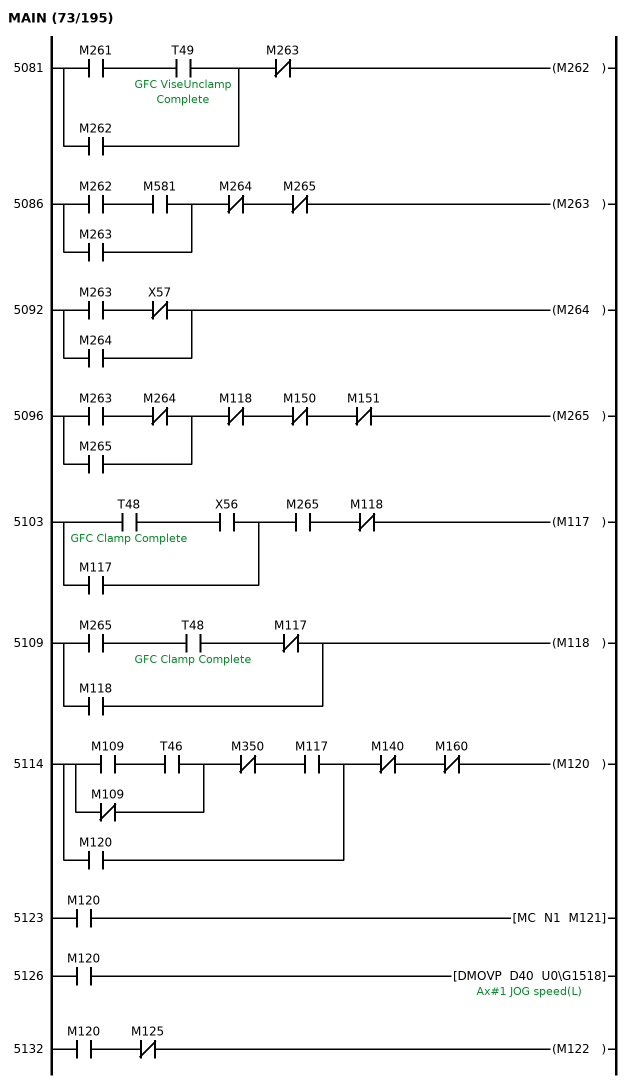
[picture p72: ladder of MAIN, rungs at steps 5081 to 5132]
5081  LD      M261
      AND     T49  ; GFC ViseUnclamp Complete
      OR      M262
      ANI     M263
      OUT     M262
5086  LD      M262
      AND     M581
      OR      M263
      ANI     M264
      ANI     M265
      OUT     M263
5092  LD      M263
      ANI     X57
      OR      M264
      OUT     M264
5096  LD      M263
      ANI     M264
      OR      M265
      ANI     M118
      ANI     M150
      ANI     M151
      OUT     M265
5103  LD      T48  ; GFC Clamp Complete
      AND     X56
      OR      M117
      AND     M265
      ANI     M118
      OUT     M117
5109  LD      M265
      AND     T48  ; GFC Clamp Complete
      ANI     M117
      OR      M118
      OUT     M118
5114  LD      M109
      AND     T46
      ORI     M109
      ANI     M350
      AND     M117
      OR      M120
      ANI     M140
      ANI     M160
      OUT     M120
5123  LD      M120
      MC      N1 M121
5126  LD      M120
      DMOVP   D40 U0\G1518
5132  LD      M120
      ANI     M125
      OUT     M122
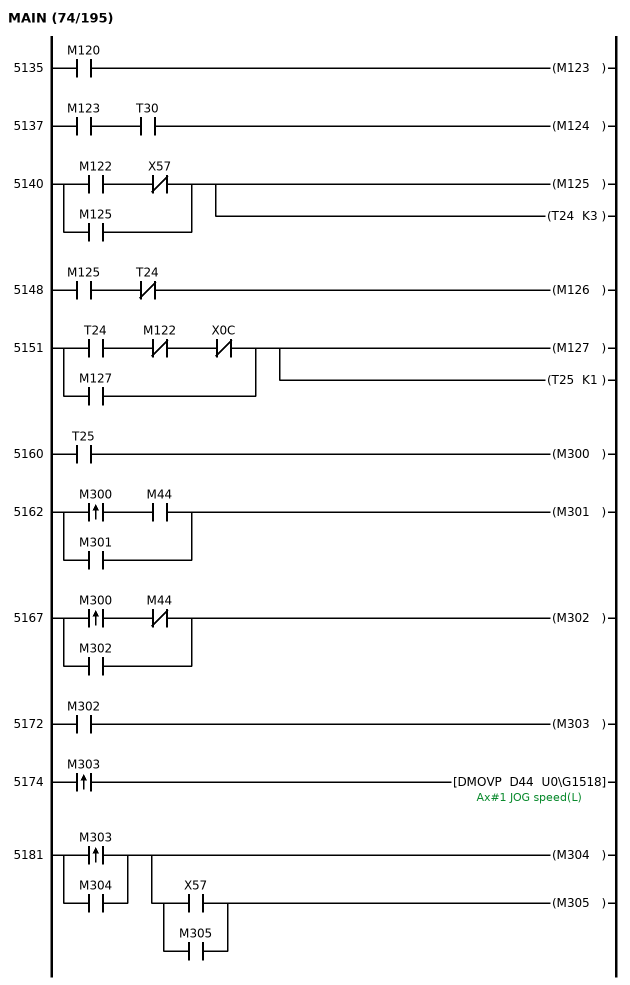
5135  LD      M120
      OUT     M123
5137  LD      M123
      AND     T30
      OUT     M124
5140  LD      M122
      ANI     X57
      OR      M125
      OUT     M125
      OUT     T24 K3
5148  LD      M125
      ANI     T24
      OUT     M126
5151  LD      T24
      ANI     M122
      ANI     X0C
      OR      M127
      OUT     M127
      OUT     T25 K1
5160  LD      T25
      OUT     M300
5162  LDP     M300
      AND     M44
      OR      M301
      OUT     M301
5167  LDP     M300
      ANI     M44
      OR      M302
      OUT     M302
5172  LD      M302
      OUT     M303
5174  LDP     M303
      DMOVP   D44 U0\G1518
5181  LDP     M303
      OR      M304
      OUT     M304
      LD      X57
      OR      M305
      ANB
      OUT     M305
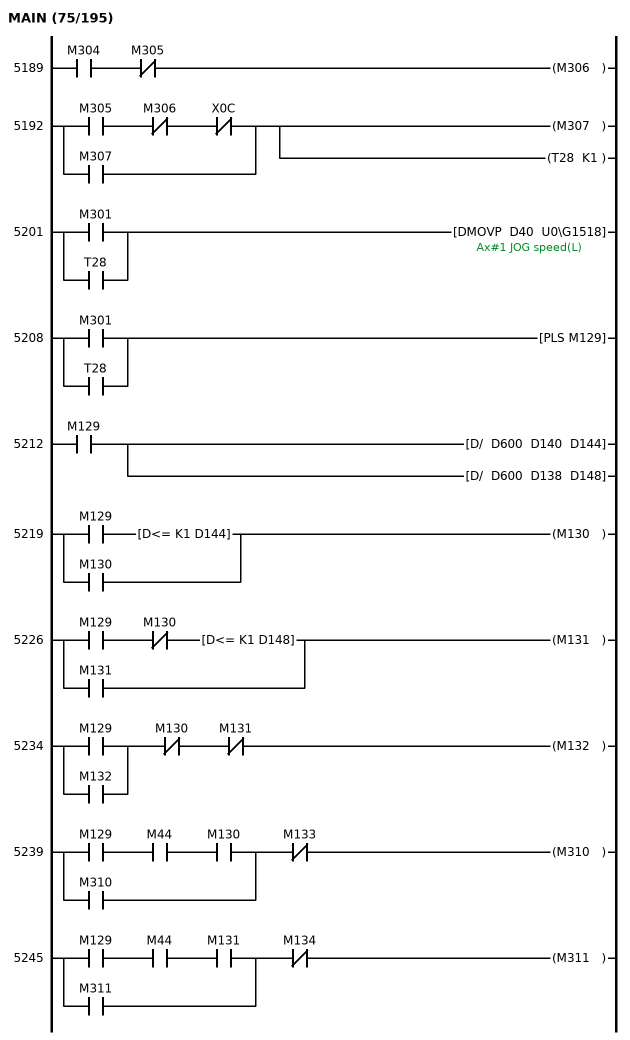
5189  LD      M304
      ANI     M305
      OUT     M306
5192  LD      M305
      ANI     M306
      ANI     X0C
      OR      M307
      OUT     M307
      OUT     T28 K1
5201  LD      M301
      OR      T28
      DMOVP   D40 U0\G1518
5208  LD      M301
      OR      T28
      PLS     M129
5212  LD      M129
      D/      D600 D140 D144
      D/      D600 D138 D148
5219  LD      M129
      ANDD<=  K1 D144
      OR      M130
      OUT     M130
5226  LD      M129
      ANI     M130
      ANDD<=  K1 D148
      OR      M131
      OUT     M131
5234  LD      M129
      OR      M132
      ANI     M130
      ANI     M131
      OUT     M132
5239  LD      M129
      AND     M44
      AND     M130
      OR      M310
      ANI     M133
      OUT     M310
5245  LD      M129
      AND     M44
      AND     M131
      OR      M311
      ANI     M134
      OUT     M311
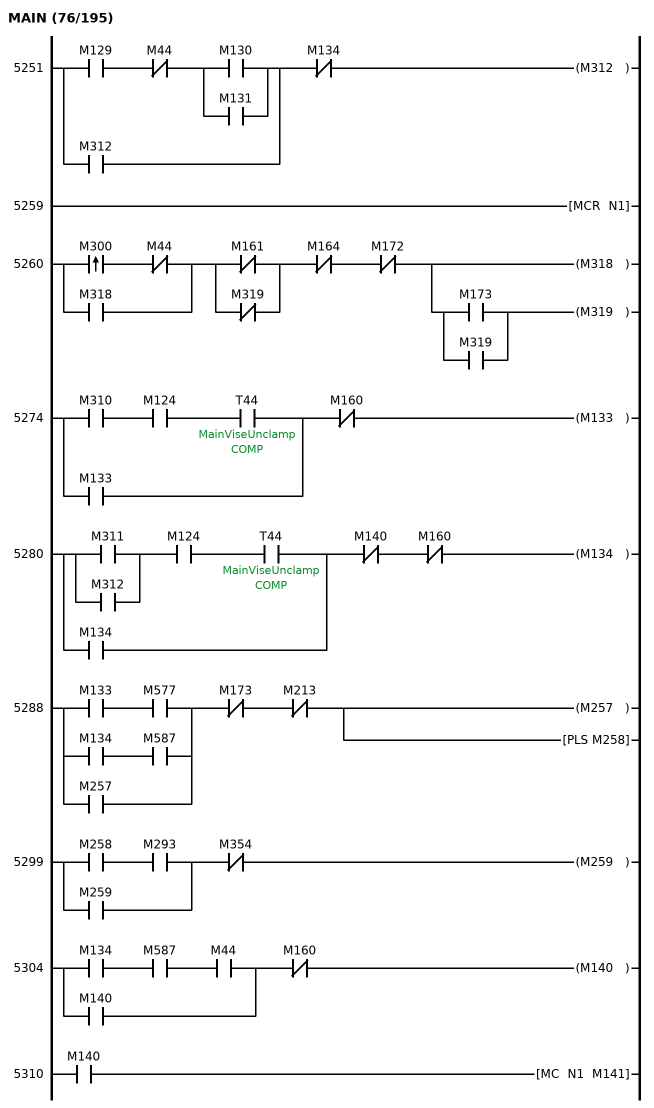
5251  LD      M129
      ANI     M44
      LD      M130
      OR      M131
      ANB
      OR      M312
      ANI     M134
      OUT     M312
5259  MCR     N1
5260  LDP     M300
      ANI     M44
      OR      M318
      LDI     M161
      ORI     M319
      ANB
      ANI     M164
      ANI     M172
      OUT     M318
      LD      M173
      OR      M319
      ANB
      OUT     M319
5274  LD      M310
      AND     M124
      AND     T44  ; MainViseUnclamp COMP
      OR      M133
      ANI     M160
      OUT     M133
5280  LD      M311
      OR      M312
      AND     M124
      AND     T44  ; MainViseUnclamp COMP
      OR      M134
      ANI     M140
      ANI     M160
      OUT     M134
5288  LD      M133
      AND     M577
      LD      M134
      AND     M587
      ORB
      OR      M257
      ANI     M173
      ANI     M213
      OUT     M257
      PLS     M258
5299  LD      M258
      AND     M293
      OR      M259
      ANI     M354
      OUT     M259
5304  LD      M134
      AND     M587
      AND     M44
      OR      M140
      ANI     M160
      OUT     M140
5310  LD      M140
      MC      N1 M141
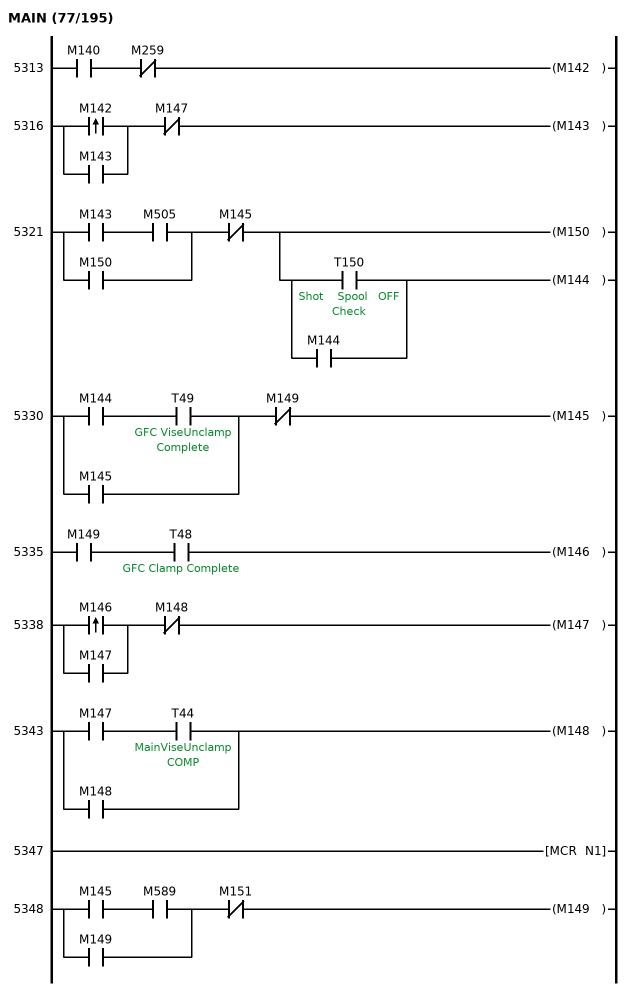
5313  LD      M140
      ANI     M259
      OUT     M142
5316  LDP     M142
      OR      M143
      ANI     M147
      OUT     M143
5321  LD      M143
      AND     M505
      OR      M150
      ANI     M145
      OUT     M150
      LD      T150  ; Shot    Spool   OFF     Check
      OR      M144
      ANB
      OUT     M144
5330  LD      M144
      AND     T49  ; GFC ViseUnclamp Complete
      OR      M145
      ANI     M149
      OUT     M145
5335  LD      M149
      AND     T48  ; GFC Clamp Complete
      OUT     M146
5338  LDP     M146
      OR      M147
      ANI     M148
      OUT     M147
5343  LD      M147
      AND     T44  ; MainViseUnclamp COMP
      OR      M148
      OUT     M148
5347  MCR     N1
5348  LD      M145
      AND     M589
      OR      M149
      ANI     M151
      OUT     M149
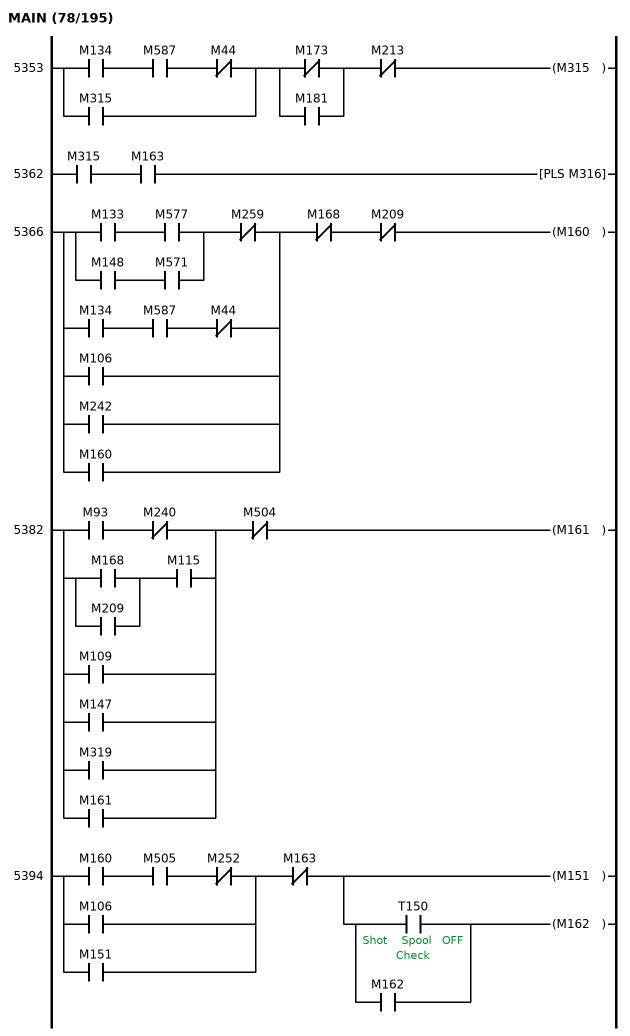
5353  LD      M134
      AND     M587
      ANI     M44
      OR      M315
      LDI     M173
      OR      M181
      ANB
      ANI     M213
      OUT     M315
5362  LD      M315
      AND     M163
      PLS     M316
5366  LD      M133
      AND     M577
      LD      M148
      AND     M571
      ORB
      ANI     M259
      LD      M134
      AND     M587
      ANI     M44
      ORB
      OR      M106
      OR      M242
      OR      M160
      ANI     M168
      ANI     M209
      OUT     M160
5382  LD      M93
      ANI     M240
      LD      M168
      OR      M209
      AND     M115
      ORB
      OR      M109
      OR      M147
      OR      M319
      OR      M161
      ANI     M504
      OUT     M161
5394  LD      M160
      AND     M505
      ANI     M252
      OR      M106
      OR      M151
      ANI     M163
      OUT     M151
      LD      T150  ; Shot    Spool   OFF     Check
      OR      M162
      ANB
      OUT     M162
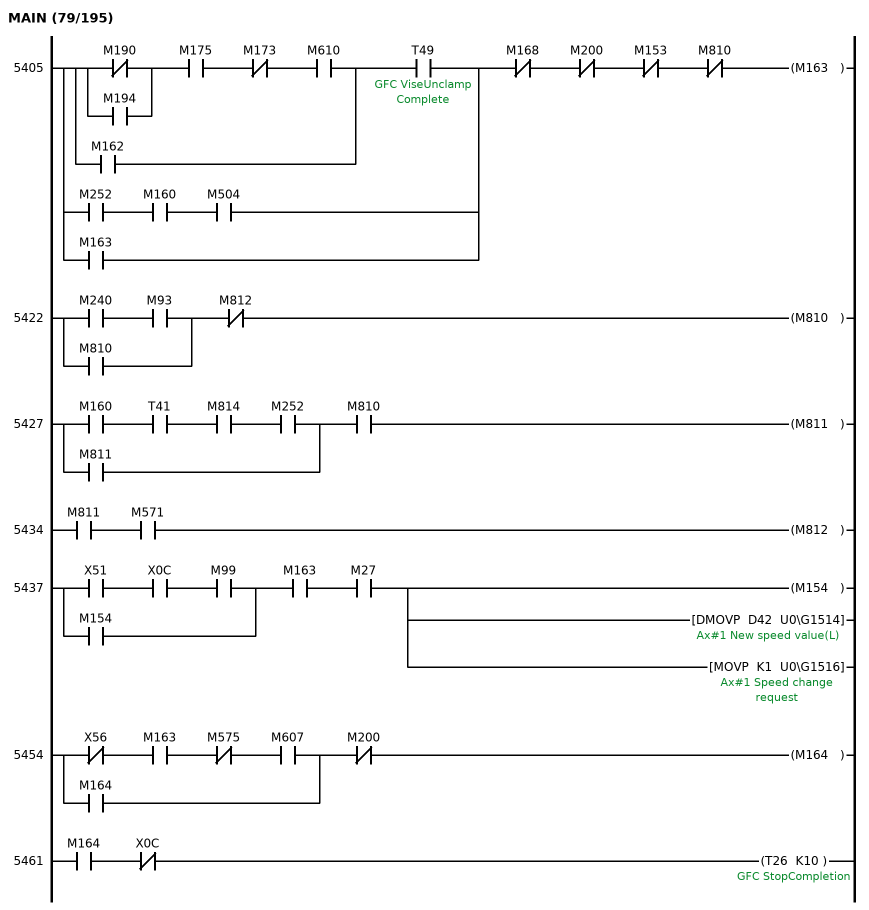
5405  LDI     M190
      OR      M194
      AND     M175
      ANI     M173
      AND     M610
      OR      M162
      AND     T49  ; GFC ViseUnclamp Complete
      LD      M252
      AND     M160
      AND     M504
      ORB
      OR      M163
      ANI     M168
      ANI     M200
      ANI     M153
      ANI     M810
      OUT     M163
5422  LD      M240
      AND     M93
      OR      M810
      ANI     M812
      OUT     M810
5427  LD      M160
      AND     T41
      AND     M814
      AND     M252
      OR      M811
      AND     M810
      OUT     M811
5434  LD      M811
      AND     M571
      OUT     M812
5437  LD      X51
      AND     X0C
      AND     M99
      OR      M154
      AND     M163
      AND     M27
      OUT     M154
      DMOVP   D42 U0\G1514  ; Ax#1 New speed value(L)
      MOVP    K1 U0\G1516  ; Ax#1 Speed change request
5454  LDI     X56
      AND     M163
      ANI     M575
      AND     M607
      OR      M164
      ANI     M200
      OUT     M164
5461  LD      M164
      ANI     X0C
      OUT     T26 K10  ; GFC StopCompletion
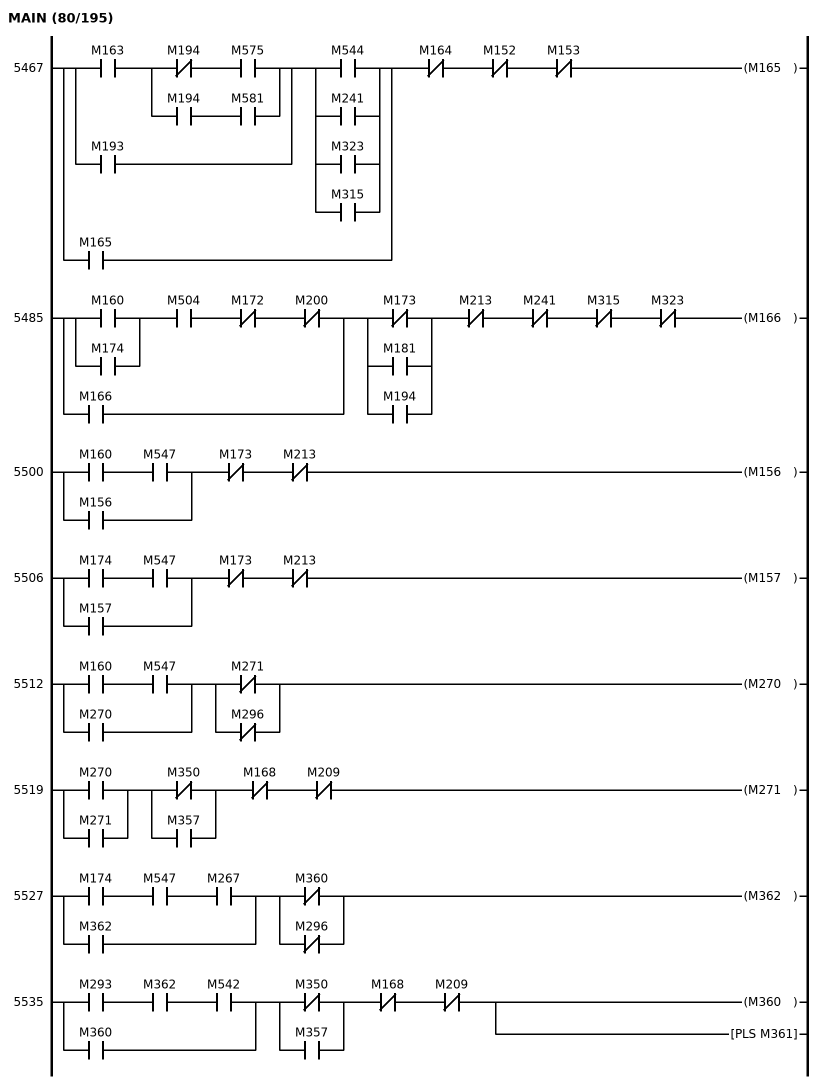
5467  LD      M163
      LDI     M194
      AND     M575
      LD      M194
      AND     M581
      ORB
      ANB
      OR      M193
      LD      M544
      OR      M241
      OR      M323
      OR      M315
      ANB
      OR      M165
      ANI     M164
      ANI     M152
      ANI     M153
      OUT     M165
5485  LD      M160
      OR      M174
      AND     M504
      ANI     M172
      ANI     M200
      OR      M166
      LDI     M173
      OR      M181
      OR      M194
      ANB
      ANI     M213
      ANI     M241
      ANI     M315
      ANI     M323
      OUT     M166
5500  LD      M160
      AND     M547
      OR      M156
      ANI     M173
      ANI     M213
      OUT     M156
5506  LD      M174
      AND     M547
      OR      M157
      ANI     M173
      ANI     M213
      OUT     M157
5512  LD      M160
      AND     M547
      OR      M270
      LDI     M271
      ORI     M296
      ANB
      OUT     M270
5519  LD      M270
      OR      M271
      LDI     M350
      OR      M357
      ANB
      ANI     M168
      ANI     M209
      OUT     M271
5527  LD      M174
      AND     M547
      AND     M267
      OR      M362
      LDI     M360
      ORI     M296
      ANB
      OUT     M362
5535  LD      M293
      AND     M362
      AND     M542
      OR      M360
      LDI     M350
      OR      M357
      ANB
      ANI     M168
      ANI     M209
      OUT     M360
      PLS     M361
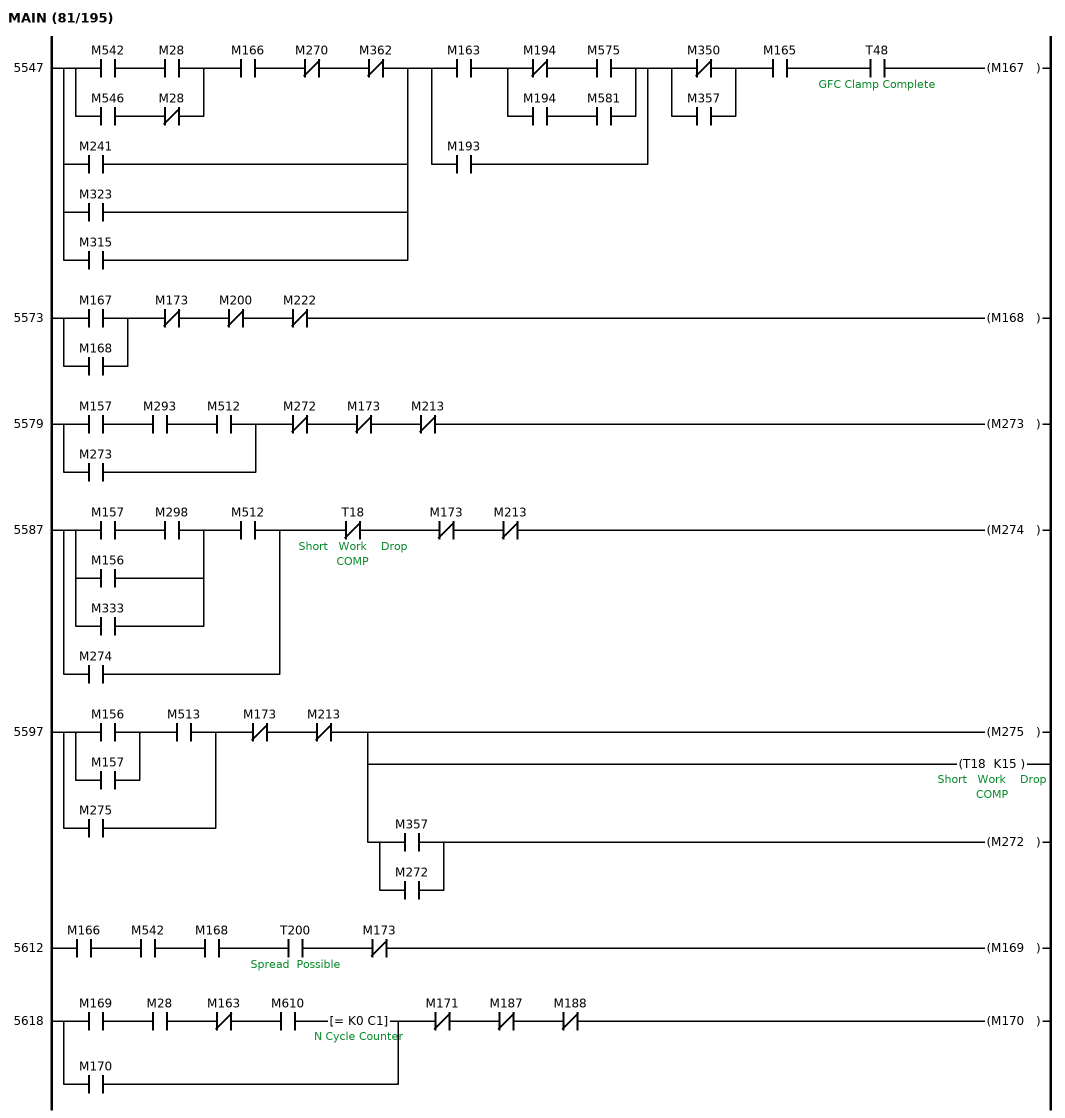
5547  LD      M542
      AND     M28
      LD      M546
      ANI     M28
      ORB
      AND     M166
      ANI     M270
      ANI     M362
      OR      M241
      OR      M323
      OR      M315
      LD      M163
      LDI     M194
      AND     M575
      LD      M194
      AND     M581
      ORB
      ANB
      OR      M193
      ANB
      LDI     M350
      OR      M357
      ANB
      AND     M165
      AND     T48  ; GFC Clamp Complete
      OUT     M167
5573  LD      M167
      OR      M168
      ANI     M173
      ANI     M200
      ANI     M222
      OUT     M168
5579  LD      M157
      AND     M293
      AND     M512
      OR      M273
      ANI     M272
      ANI     M173
      ANI     M213
      OUT     M273
5587  LD      M157
      AND     M298
      OR      M156
      OR      M333
      AND     M512
      OR      M274
      ANI     T18  ; Short   Work    Drop    COMP
      ANI     M173
      ANI     M213
      OUT     M274
5597  LD      M156
      OR      M157
      AND     M513
      OR      M275
      ANI     M173
      ANI     M213
      OUT     M275
      OUT     T18 K15  ; Short   Work    Drop    COMP
      LD      M357
      OR      M272
      ANB
      OUT     M272
5612  LD      M166
      AND     M542
      AND     M168
      AND     T200  ; Spread  Possible
      ANI     M173
      OUT     M169
5618  LD      M169
      AND     M28
      ANI     M163
      AND     M610
      AND=    K0 C1  ; N Cycle Counter
      OR      M170
      ANI     M171
      ANI     M187
      ANI     M188
      OUT     M170
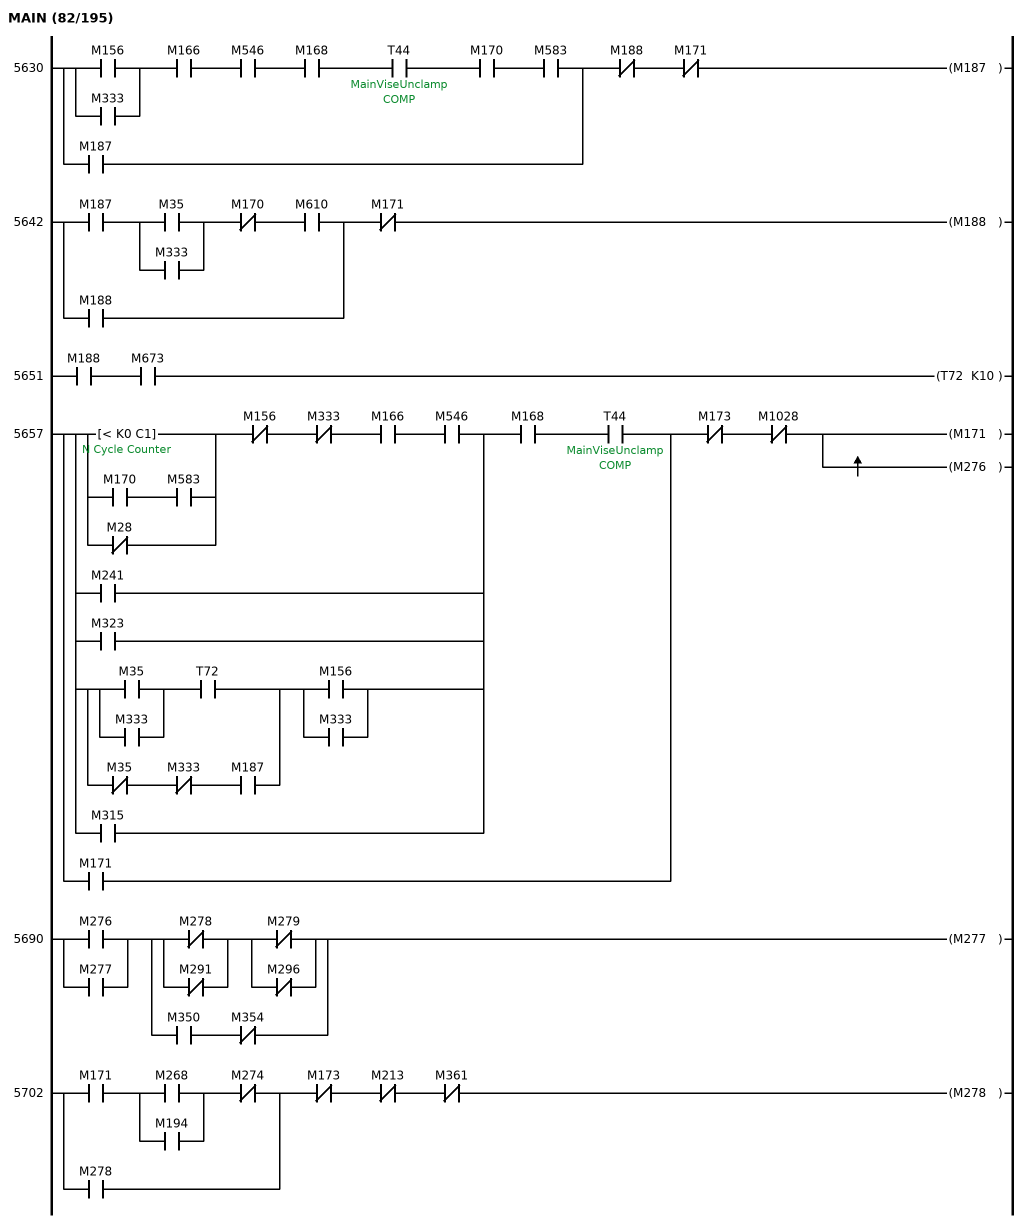
5630  LD      M156
      OR      M333
      AND     M166
      AND     M546
      AND     M168
      AND     T44  ; MainViseUnclamp COMP
      AND     M170
      AND     M583
      OR      M187
      ANI     M188
      ANI     M171
      OUT     M187
5642  LD      M187
      LD      M35
      OR      M333
      ANB
      ANI     M170
      AND     M610
      OR      M188
      ANI     M171
      OUT     M188
5651  LD      M188
      AND     M673
      OUT     T72 K10
5657  LD<     K0 C1  ; N Cycle Counter
      LD      M170
      AND     M583
      ORB
      ORI     M28
      ANI     M156
      ANI     M333
      AND     M166
      AND     M546
      OR      M241
      OR      M323
      LD      M35
      OR      M333
      AND     T72
      LDI     M35
      ANI     M333
      AND     M187
      ORB
      LD      M156
      OR      M333
      ANB
      ORB
      OR      M315
      AND     M168
      AND     T44  ; MainViseUnclamp COMP
      OR      M171
      ANI     M173
      ANI     M1028
      OUT     M171
      MEP
      OUT     M276
5690  LD      M276
      OR      M277
      LDI     M278
      ORI     M291
      LDI     M279
      ORI     M296
      ANB
      LD      M350
      ANI     M354
      ORB
      ANB
      OUT     M277
5702  LD      M171
      LD      M268
      OR      M194
      ANB
      ANI     M274
      OR      M278
      ANI     M173
      ANI     M213
      ANI     M361
      OUT     M278
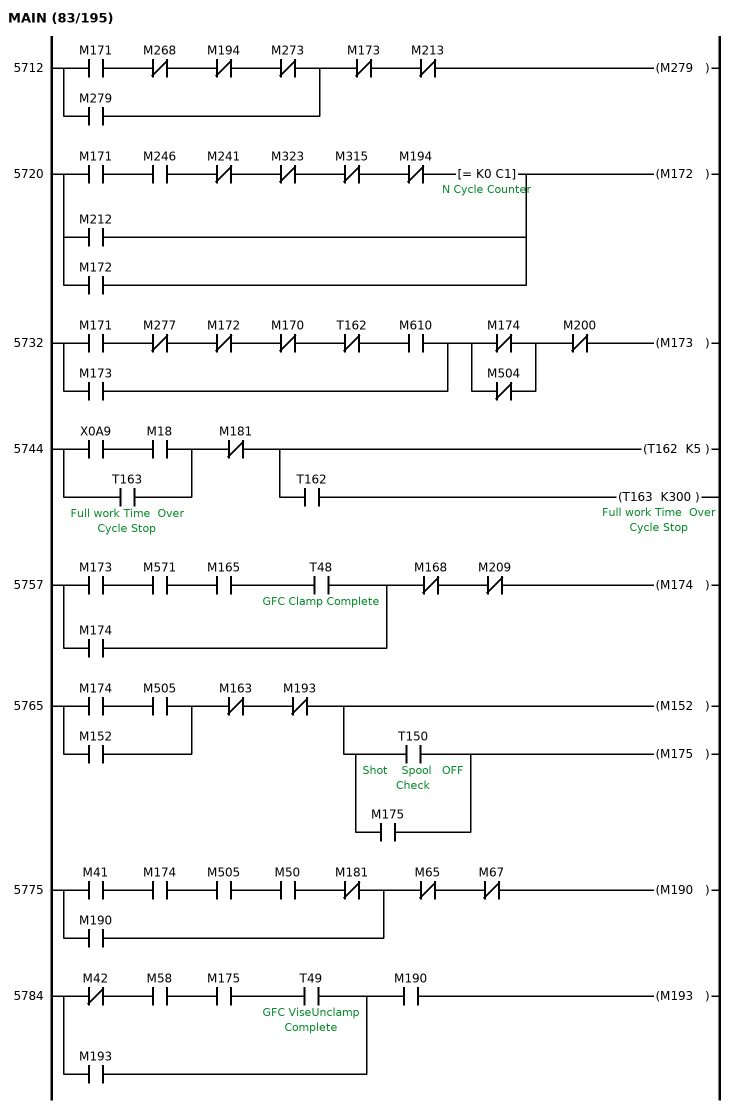
5712  LD      M171
      ANI     M268
      ANI     M194
      ANI     M273
      OR      M279
      ANI     M173
      ANI     M213
      OUT     M279
5720  LD      M171
      AND     M246
      ANI     M241
      ANI     M323
      ANI     M315
      ANI     M194
      AND=    K0 C1  ; N Cycle Counter
      OR      M212
      OR      M172
      OUT     M172
5732  LD      M171
      ANI     M277
      ANI     M172
      ANI     M170
      ANI     T162
      AND     M610
      OR      M173
      LDI     M174
      ORI     M504
      ANB
      ANI     M200
      OUT     M173
5744  LD      X0A9
      AND     M18
      OR      T163  ; Full work Time  Over Cycle Stop
      ANI     M181
      OUT     T162 K5
      AND     T162
      OUT     T163 K300  ; Full work Time  Over Cycle Stop
5757  LD      M173
      AND     M571
      AND     M165
      AND     T48  ; GFC Clamp Complete
      OR      M174
      ANI     M168
      ANI     M209
      OUT     M174
5765  LD      M174
      AND     M505
      OR      M152
      ANI     M163
      ANI     M193
      OUT     M152
      LD      T150  ; Shot    Spool   OFF     Check
      OR      M175
      ANB
      OUT     M175
5775  LD      M41
      AND     M174
      AND     M505
      AND     M50
      ANI     M181
      OR      M190
      ANI     M65
      ANI     M67
      OUT     M190
5784  LDI     M42
      AND     M58
      AND     M175
      AND     T49  ; GFC ViseUnclamp Complete
      OR      M193
      AND     M190
      OUT     M193
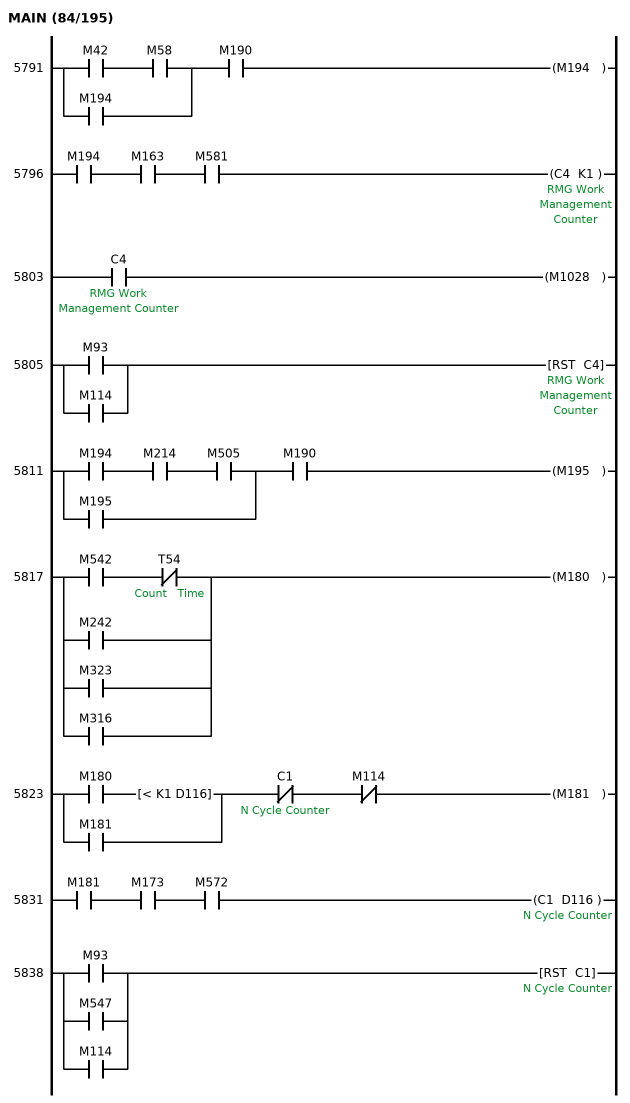
5791  LD      M42
      AND     M58
      OR      M194
      AND     M190
      OUT     M194
5796  LD      M194
      AND     M163
      AND     M581
      OUT     C4 K1  ; RMG WorkManagement Counter
5803  LD      C4  ; RMG WorkManagement Counter
      OUT     M1028
5805  LD      M93
      OR      M114
      RST     C4  ; RMG WorkManagement Counter
5811  LD      M194
      AND     M214
      AND     M505
      OR      M195
      AND     M190
      OUT     M195
5817  LD      M542
      ANI     T54  ; Count   Time
      OR      M242
      OR      M323
      OR      M316
      OUT     M180
5823  LD      M180
      AND<    K1 D116
      OR      M181
      ANI     C1  ; N Cycle Counter
      ANI     M114
      OUT     M181
5831  LD      M181
      AND     M173
      AND     M572
      OUT     C1 D116  ; N Cycle Counter
5838  LD      M93
      OR      M547
      OR      M114
      RST     C1  ; N Cycle Counter
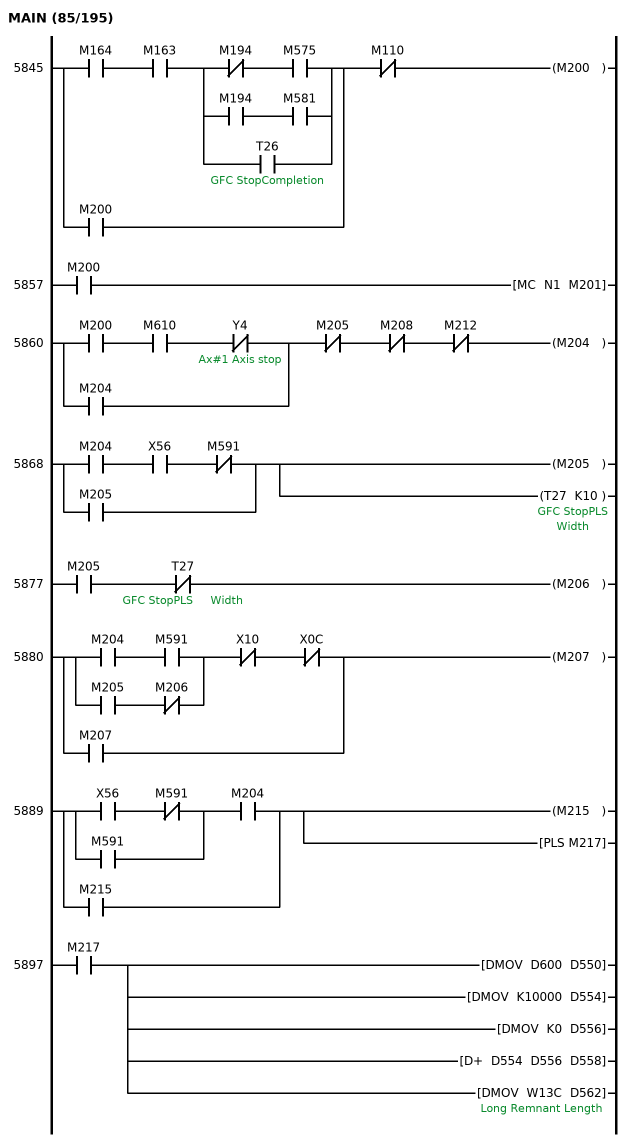
5845  LD      M164
      AND     M163
      LDI     M194
      AND     M575
      LD      M194
      AND     M581
      ORB
      OR      T26  ; GFC StopCompletion
      ANB
      OR      M200
      ANI     M110
      OUT     M200
5857  LD      M200
      MC      N1 M201
5860  LD      M200
      AND     M610
      ANI     Y4  ; Ax#1 Axis stop
      OR      M204
      ANI     M205
      ANI     M208
      ANI     M212
      OUT     M204
5868  LD      M204
      AND     X56
      ANI     M591
      OR      M205
      OUT     M205
      OUT     T27 K10  ; GFC StopPLS     Width
5877  LD      M205
      ANI     T27  ; GFC StopPLS     Width
      OUT     M206
5880  LD      M204
      AND     M591
      LD      M205
      ANI     M206
      ORB
      ANI     X10
      ANI     X0C
      OR      M207
      OUT     M207
5889  LD      X56
      ANI     M591
      OR      M591
      AND     M204
      OR      M215
      OUT     M215
      PLS     M217
5897  LD      M217
      DMOV    D600 D550
      DMOV    K10000 D554
      DMOV    K0 D556
      D+      D554 D556 D558
      DMOV    W13C D562  ; Long Remnant Length
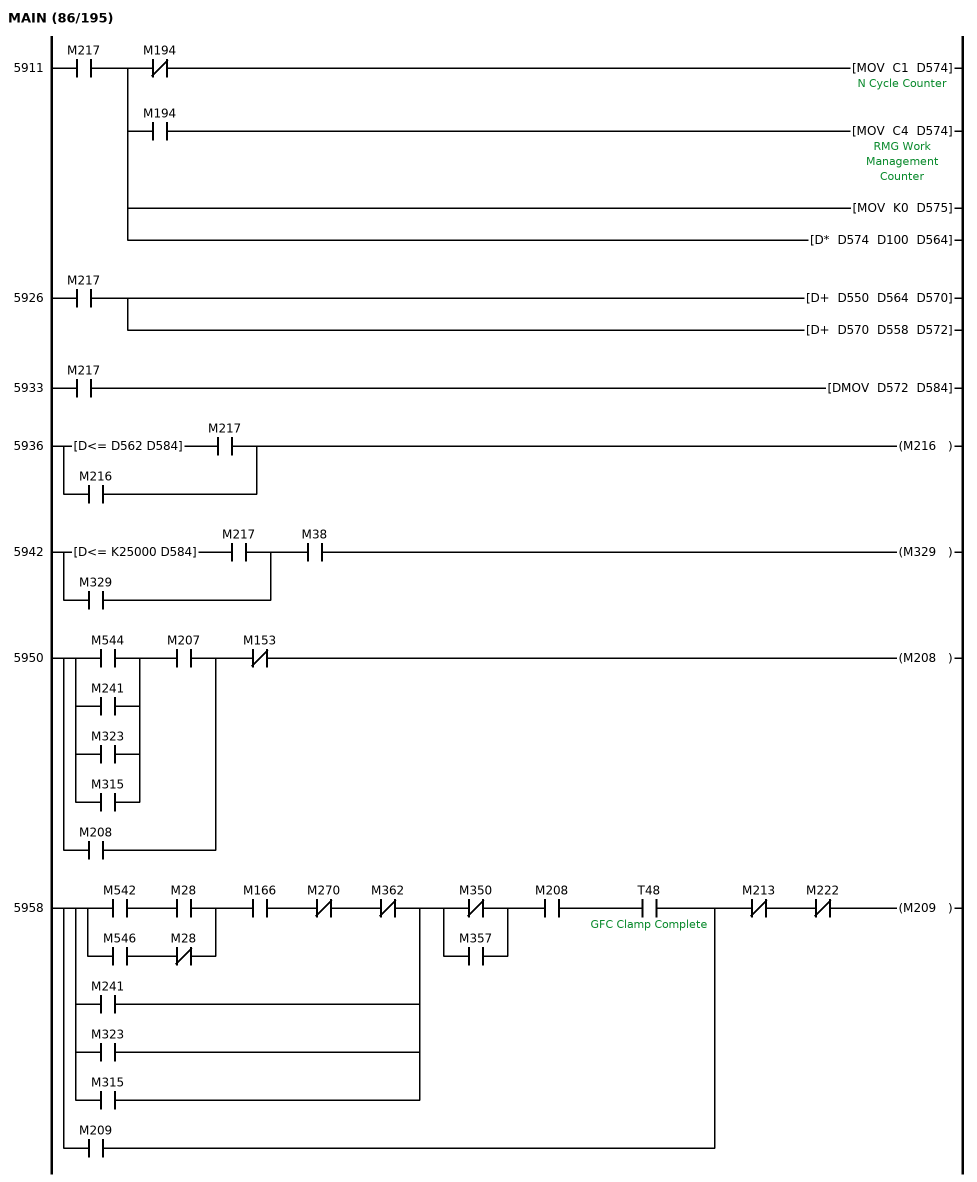
5911  LD      M217
      MPS
      ANI     M194
      MOV     C1 D574
      MRD
      AND     M194
      MOV     C4 D574
      MPP
      MOV     K0 D575
      D*      D574 D100 D564
5926  LD      M217
      D+      D550 D564 D570
      D+      D570 D558 D572
5933  LD      M217
      DMOV    D572 D584
5936  LDD<=   D562 D584
      AND     M217
      OR      M216
      OUT     M216
5942  LDD<=   K25000 D584
      AND     M217
      OR      M329
      AND     M38
      OUT     M329
5950  LD      M544
      OR      M241
      OR      M323
      OR      M315
      AND     M207
      OR      M208
      ANI     M153
      OUT     M208
5958  LD      M542
      AND     M28
      LD      M546
      ANI     M28
      ORB
      AND     M166
      ANI     M270
      ANI     M362
      OR      M241
      OR      M323
      OR      M315
      LDI     M350
      OR      M357
      ANB
      AND     M208
      AND     T48  ; GFC Clamp Complete
      OR      M209
      ANI     M213
      ANI     M222
      OUT     M209
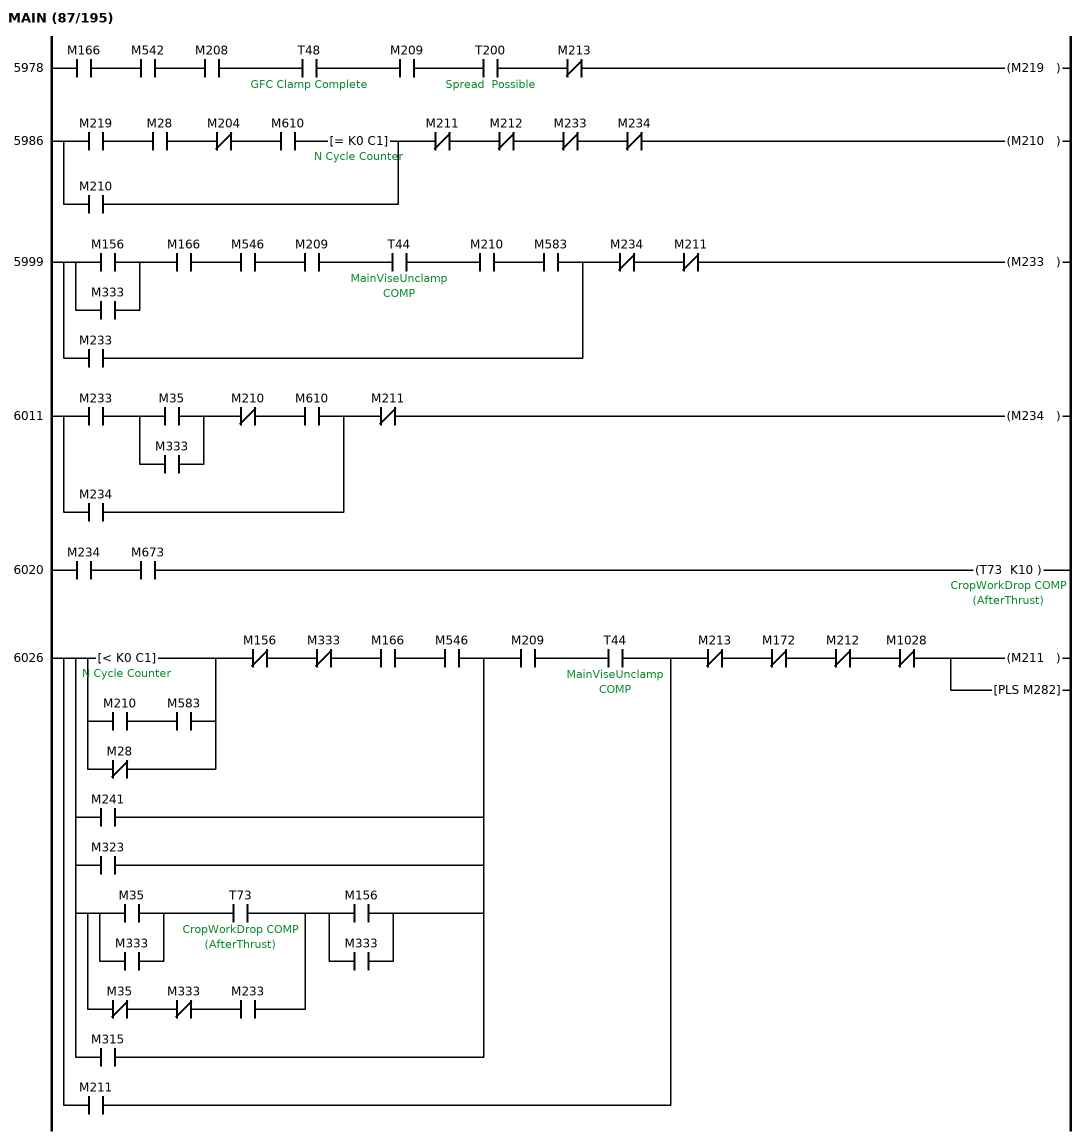
5978  LD      M166
      AND     M542
      AND     M208
      AND     T48  ; GFC Clamp Complete
      AND     M209
      AND     T200  ; Spread  Possible
      ANI     M213
      OUT     M219
5986  LD      M219
      AND     M28
      ANI     M204
      AND     M610
      AND=    K0 C1  ; N Cycle Counter
      OR      M210
      ANI     M211
      ANI     M212
      ANI     M233
      ANI     M234
      OUT     M210
5999  LD      M156
      OR      M333
      AND     M166
      AND     M546
      AND     M209
      AND     T44  ; MainViseUnclamp COMP
      AND     M210
      AND     M583
      OR      M233
      ANI     M234
      ANI     M211
      OUT     M233
6011  LD      M233
      LD      M35
      OR      M333
      ANB
      ANI     M210
      AND     M610
      OR      M234
      ANI     M211
      OUT     M234
6020  LD      M234
      AND     M673
      OUT     T73 K10  ; CropWorkDrop COMP (AfterThrust)
6026  LD<     K0 C1  ; N Cycle Counter
      LD      M210
      AND     M583
      ORB
      ORI     M28
      ANI     M156
      ANI     M333
      AND     M166
      AND     M546
      OR      M241
      OR      M323
      LD      M35
      OR      M333
      AND     T73  ; CropWorkDrop COMP (AfterThrust)
      LDI     M35
      ANI     M333
      AND     M233
      ORB
      LD      M156
      OR      M333
      ANB
      ORB
      OR      M315
      AND     M209
      AND     T44  ; MainViseUnclamp COMP
      OR      M211
      ANI     M213
      ANI     M172
      ANI     M212
      ANI     M1028
      OUT     M211
      PLS     M282
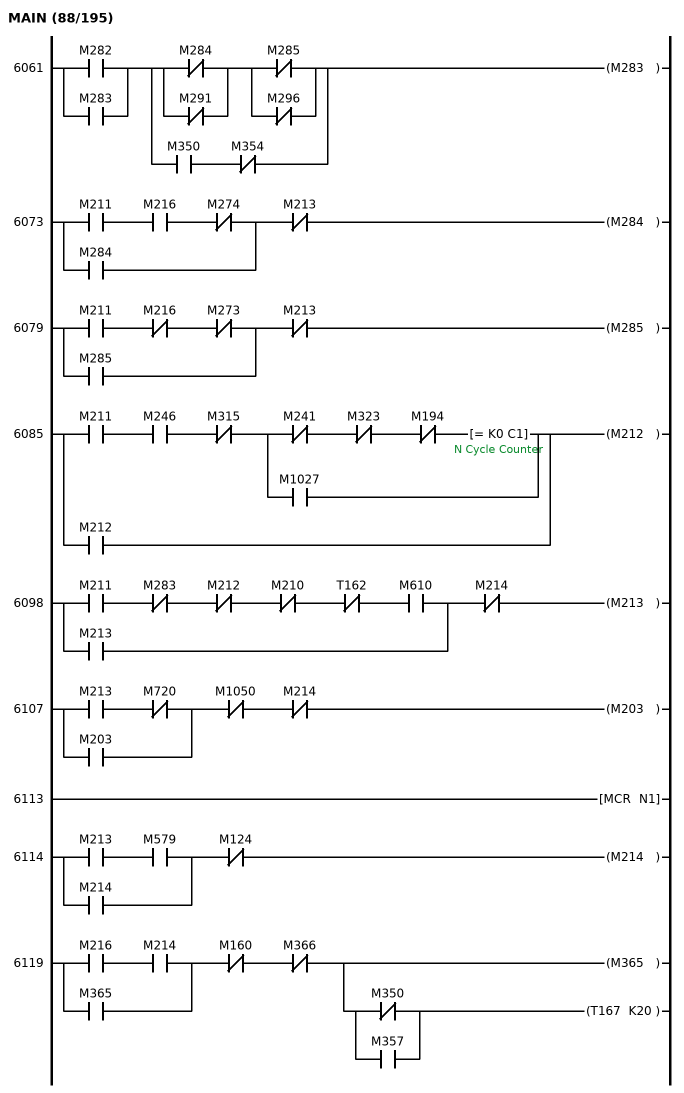
6061  LD      M282
      OR      M283
      LDI     M284
      ORI     M291
      LDI     M285
      ORI     M296
      ANB
      LD      M350
      ANI     M354
      ORB
      ANB
      OUT     M283
6073  LD      M211
      AND     M216
      ANI     M274
      OR      M284
      ANI     M213
      OUT     M284
6079  LD      M211
      ANI     M216
      ANI     M273
      OR      M285
      ANI     M213
      OUT     M285
6085  LD      M211
      AND     M246
      ANI     M315
      LDI     M241
      ANI     M323
      ANI     M194
      AND=    K0 C1  ; N Cycle Counter
      OR      M1027
      ANB
      OR      M212
      OUT     M212
6098  LD      M211
      ANI     M283
      ANI     M212
      ANI     M210
      ANI     T162
      AND     M610
      OR      M213
      ANI     M214
      OUT     M213
6107  LD      M213
      ANI     M720
      OR      M203
      ANI     M1050
      ANI     M214
      OUT     M203
6113  MCR     N1
6114  LD      M213
      AND     M579
      OR      M214
      ANI     M124
      OUT     M214
6119  LD      M216
      AND     M214
      OR      M365
      ANI     M160
      ANI     M366
      OUT     M365
      LDI     M350
      OR      M357
      ANB
      OUT     T167 K20
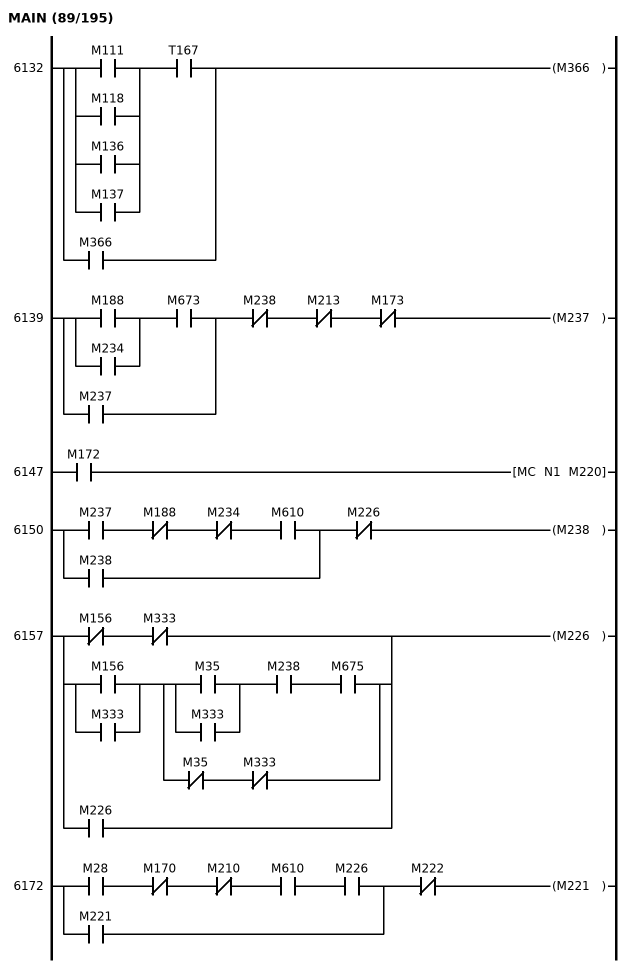
6132  LD      M111
      OR      M118
      OR      M136
      OR      M137
      AND     T167
      OR      M366
      OUT     M366
6139  LD      M188
      OR      M234
      AND     M673
      OR      M237
      ANI     M238
      ANI     M213
      ANI     M173
      OUT     M237
6147  LD      M172
      MC      N1 M220
6150  LD      M237
      ANI     M188
      ANI     M234
      AND     M610
      OR      M238
      ANI     M226
      OUT     M238
6157  LDI     M156
      ANI     M333
      LD      M156
      OR      M333
      LD      M35
      OR      M333
      AND     M238
      AND     M675
      LDI     M35
      ANI     M333
      ORB
      ANB
      ORB
      OR      M226
      OUT     M226
6172  LD      M28
      ANI     M170
      ANI     M210
      AND     M610
      AND     M226
      OR      M221
      ANI     M222
      OUT     M221
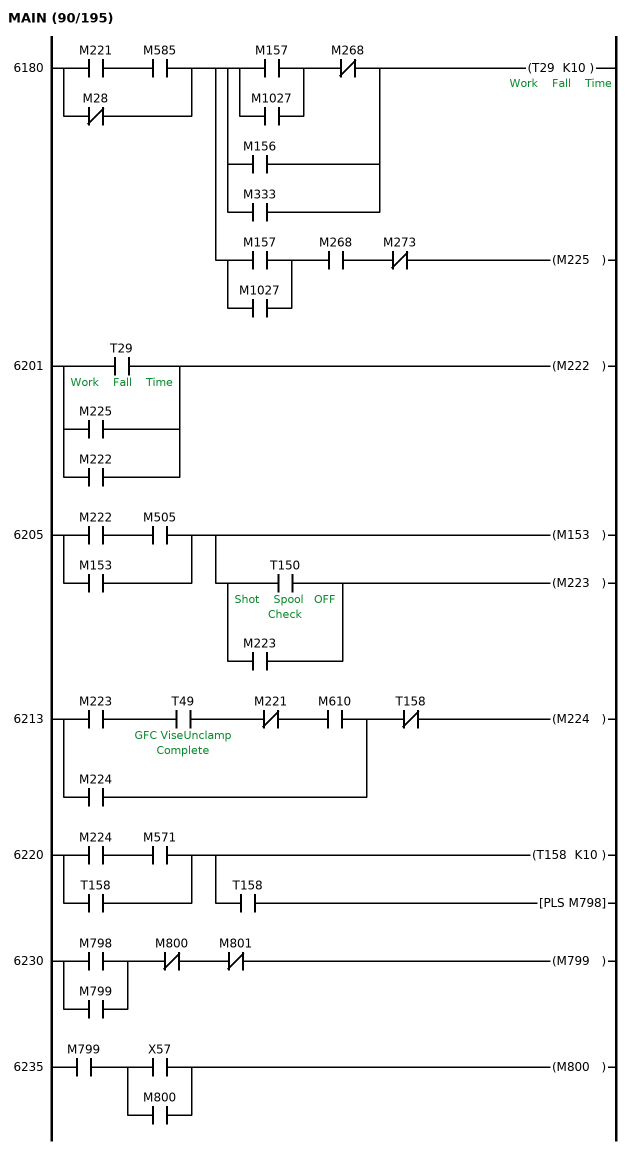
6180  LD      M221
      AND     M585
      ORI     M28
      MPS
      LD      M157
      OR      M1027
      ANI     M268
      OR      M156
      OR      M333
      ANB
      OUT     T29 K10  ; Work    Fall    Time
      MPP
      LD      M157
      OR      M1027
      ANB
      AND     M268
      ANI     M273
      OUT     M225
6201  LD      T29  ; Work    Fall    Time
      OR      M225
      OR      M222
      OUT     M222
6205  LD      M222
      AND     M505
      OR      M153
      OUT     M153
      LD      T150  ; Shot    Spool   OFF     Check
      OR      M223
      ANB
      OUT     M223
6213  LD      M223
      AND     T49  ; GFC ViseUnclamp Complete
      ANI     M221
      AND     M610
      OR      M224
      ANI     T158
      OUT     M224
6220  LD      M224
      AND     M571
      OR      T158
      OUT     T158 K10
      AND     T158
      PLS     M798
6230  LD      M798
      OR      M799
      ANI     M800
      ANI     M801
      OUT     M799
6235  LD      M799
      LD      X57
      OR      M800
      ANB
      OUT     M800
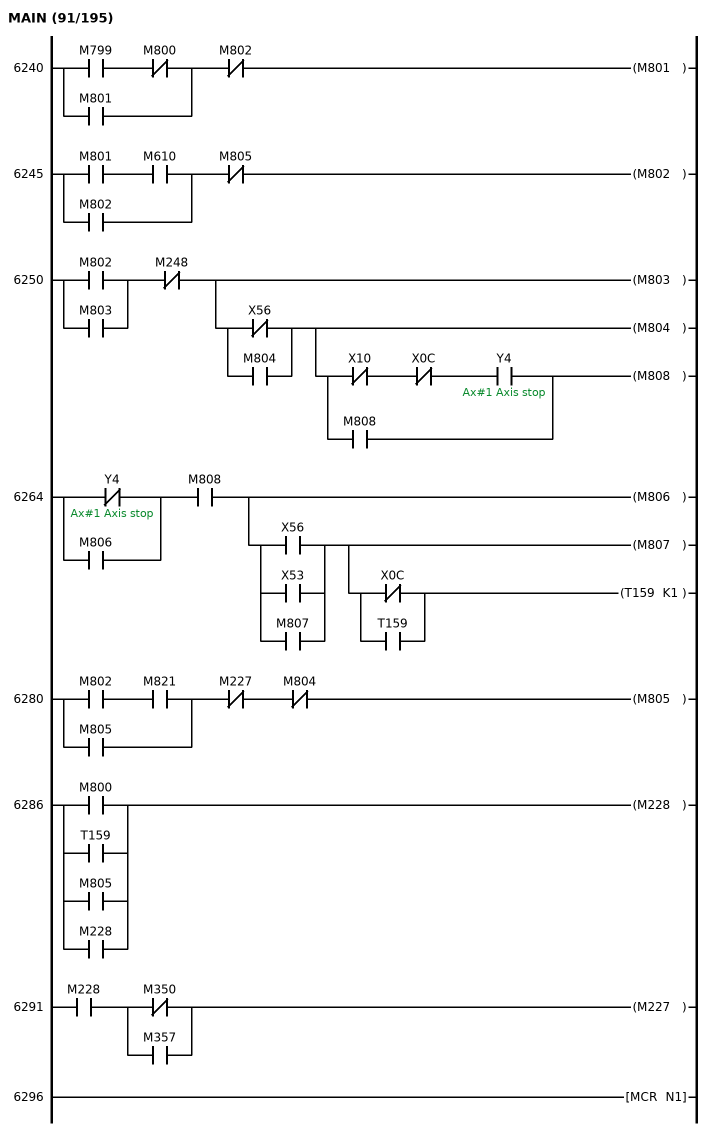
6240  LD      M799
      ANI     M800
      OR      M801
      ANI     M802
      OUT     M801
6245  LD      M801
      AND     M610
      OR      M802
      ANI     M805
      OUT     M802
6250  LD      M802
      OR      M803
      ANI     M248
      OUT     M803
      LDI     X56
      OR      M804
      ANB
      OUT     M804
      LDI     X10
      ANI     X0C
      AND     Y4  ; Ax#1 Axis stop
      OR      M808
      ANB
      OUT     M808
6264  LDI     Y4  ; Ax#1 Axis stop
      OR      M806
      AND     M808
      OUT     M806
      LD      X56
      OR      X53
      OR      M807
      ANB
      OUT     M807
      LDI     X0C
      OR      T159
      ANB
      OUT     T159 K1
6280  LD      M802
      AND     M821
      OR      M805
      ANI     M227
      ANI     M804
      OUT     M805
6286  LD      M800
      OR      T159
      OR      M805
      OR      M228
      OUT     M228
6291  LD      M228
      LDI     M350
      OR      M357
      ANB
      OUT     M227
6296  MCR     N1
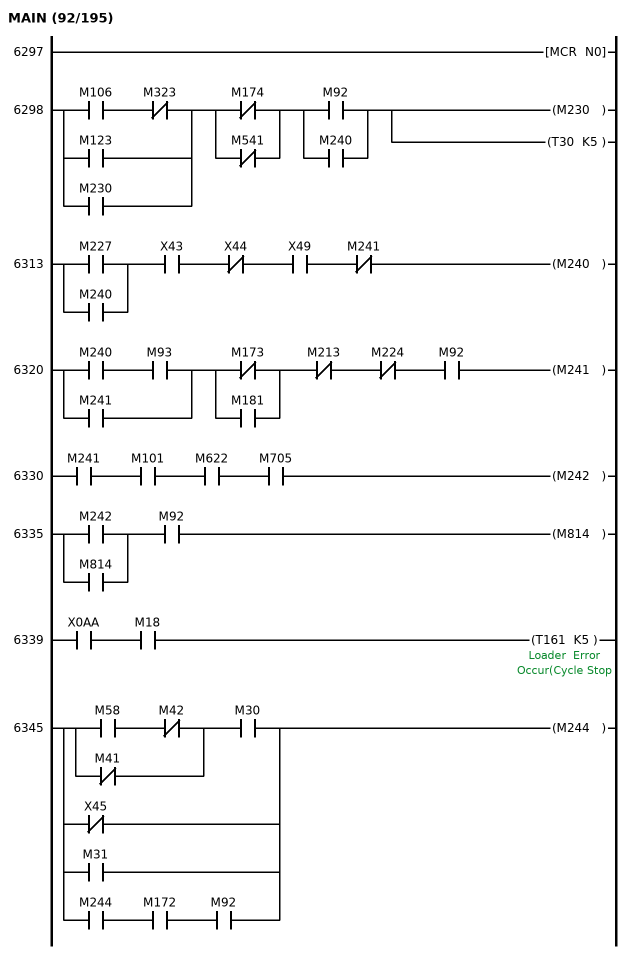
6297  MCR     N0
6298  LD      M106
      ANI     M323
      OR      M123
      OR      M230
      LDI     M174
      ORI     M541
      ANB
      LD      M92
      OR      M240
      ANB
      OUT     M230
      OUT     T30 K5
6313  LD      M227
      OR      M240
      AND     X43
      ANI     X44
      AND     X49
      ANI     M241
      OUT     M240
6320  LD      M240
      AND     M93
      OR      M241
      LDI     M173
      OR      M181
      ANB
      ANI     M213
      ANI     M224
      AND     M92
      OUT     M241
6330  LD      M241
      AND     M101
      AND     M622
      AND     M705
      OUT     M242
6335  LD      M242
      OR      M814
      AND     M92
      OUT     M814
6339  LD      X0AA
      AND     M18
      OUT     T161 K5  ; Loader  Error   Occur(Cycle Stop
6345  LD      M58
      ANI     M42
      ORI     M41
      AND     M30
      ORI     X45
      OR      M31
      LD      M244
      AND     M172
      AND     M92
      ORB
      OUT     M244
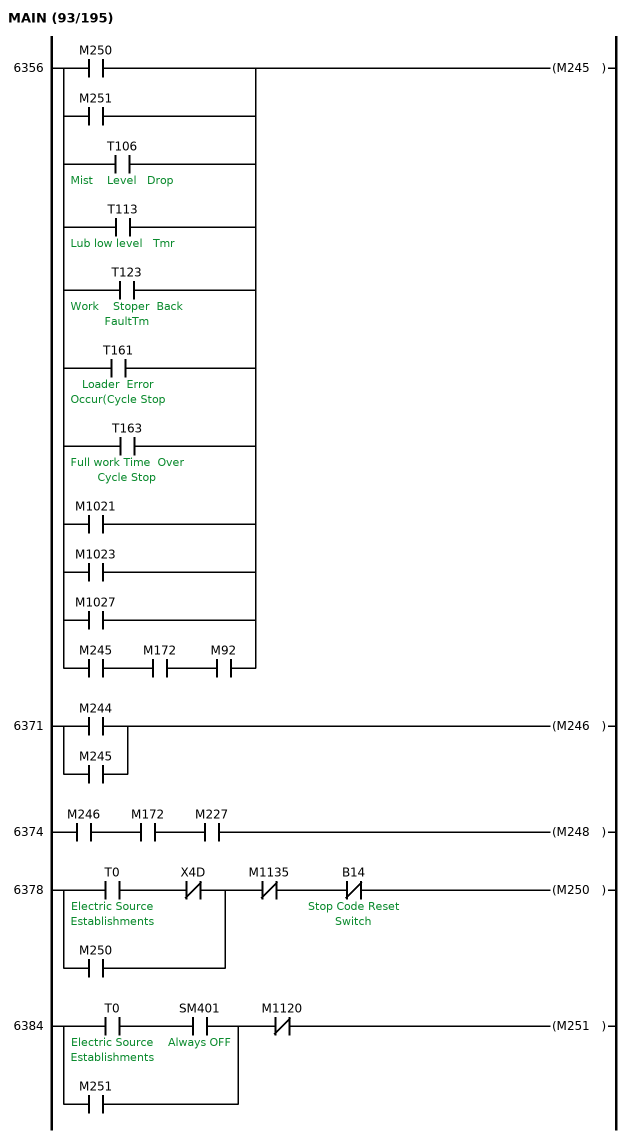
6356  LD      M250
      OR      M251
      OR      T106  ; Mist    Level   Drop
      OR      T113  ; Lub low level   Tmr
      OR      T123  ; Work    Stoper  Back    FaultTm
      OR      T161  ; Loader  Error   Occur(Cycle Stop
      OR      T163  ; Full work Time  Over Cycle Stop
      OR      M1021
      OR      M1023
      OR      M1027
      LD      M245
      AND     M172
      AND     M92
      ORB
      OUT     M245
6371  LD      M244
      OR      M245
      OUT     M246
6374  LD      M246
      AND     M172
      AND     M227
      OUT     M248
6378  LD      T0  ; Electric Source Establishments
      ANI     X4D
      OR      M250
      ANI     M1135
      ANI     B14  ; Stop Code Reset Switch
      OUT     M250
6384  LD      T0  ; Electric Source Establishments
      AND     SM401  ; Always OFF
      OR      M251
      ANI     M1120
      OUT     M251
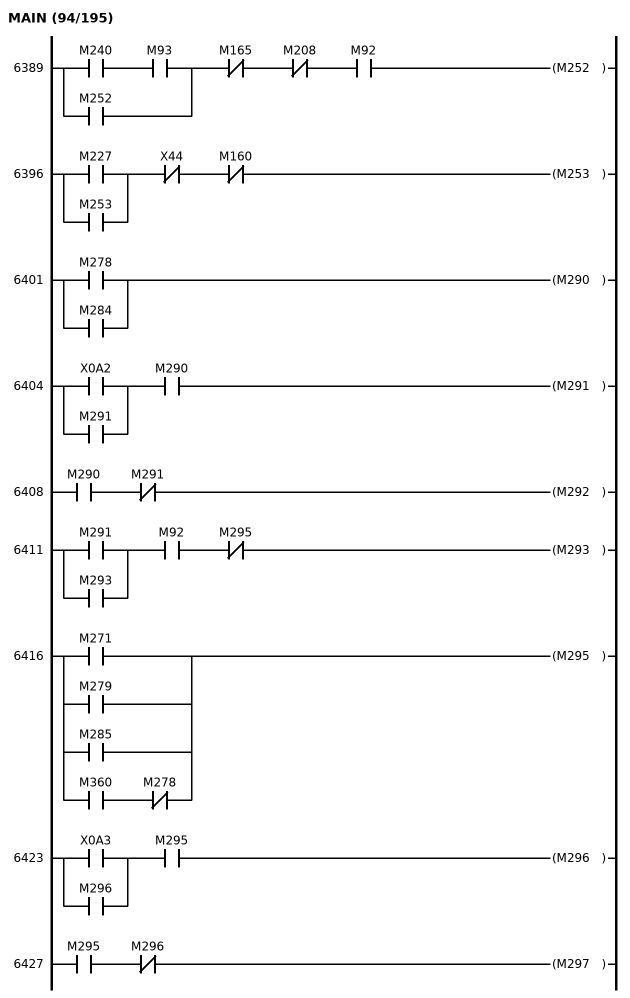
6389  LD      M240
      AND     M93
      OR      M252
      ANI     M165
      ANI     M208
      AND     M92
      OUT     M252
6396  LD      M227
      OR      M253
      ANI     X44
      ANI     M160
      OUT     M253
6401  LD      M278
      OR      M284
      OUT     M290
6404  LD      X0A2
      OR      M291
      AND     M290
      OUT     M291
6408  LD      M290
      ANI     M291
      OUT     M292
6411  LD      M291
      OR      M293
      AND     M92
      ANI     M295
      OUT     M293
6416  LD      M271
      OR      M279
      OR      M285
      LD      M360
      ANI     M278
      ORB
      OUT     M295
6423  LD      X0A3
      OR      M296
      AND     M295
      OUT     M296
6427  LD      M295
      ANI     M296
      OUT     M297
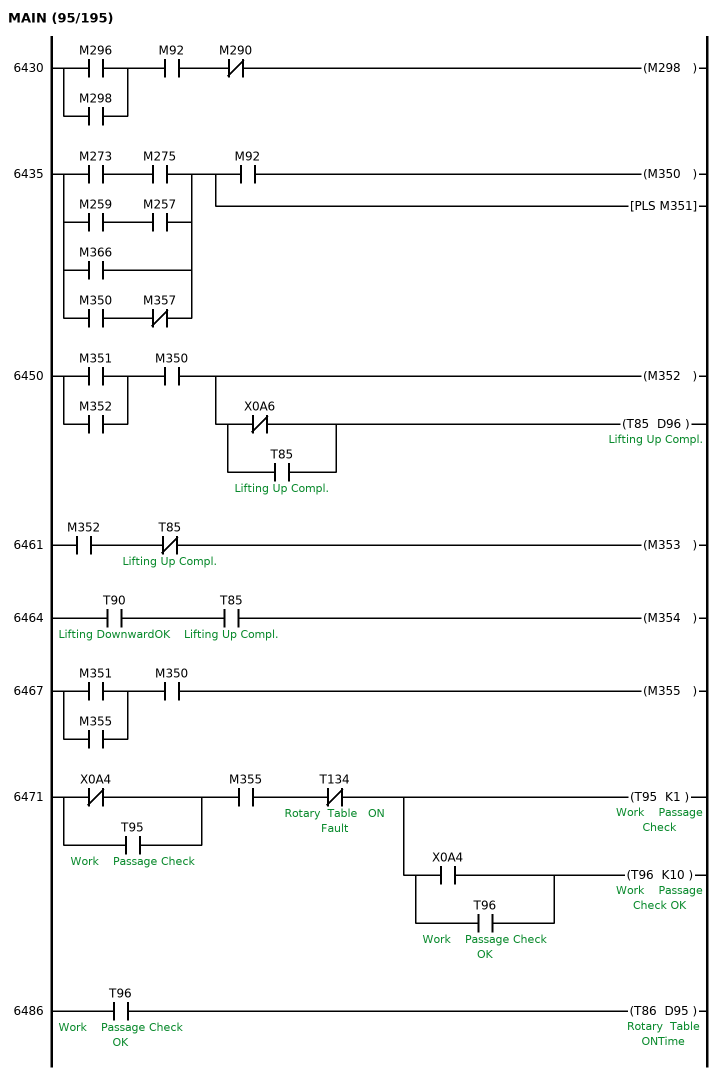
6430  LD      M296
      OR      M298
      AND     M92
      ANI     M290
      OUT     M298
6435  LD      M273
      AND     M275
      LD      M259
      AND     M257
      ORB
      OR      M366
      LD      M350
      ANI     M357
      ORB
      MPS
      AND     M92
      OUT     M350
      MPP
      PLS     M351
6450  LD      M351
      OR      M352
      AND     M350
      OUT     M352
      LDI     X0A6
      OR      T85  ; Lifting Up Compl.
      ANB
      OUT     T85 D96  ; Lifting Up Compl.
6461  LD      M352
      ANI     T85  ; Lifting Up Compl.
      OUT     M353
6464  LD      T90  ; Lifting DownwardOK
      AND     T85  ; Lifting Up Compl.
      OUT     M354
6467  LD      M351
      OR      M355
      AND     M350
      OUT     M355
6471  LDI     X0A4
      OR      T95  ; Work    Passage Check
      AND     M355
      ANI     T134  ; Rotary  Table   ON Fault
      OUT     T95 K1  ; Work    Passage Check
      LD      X0A4
      OR      T96  ; Work    Passage Check OK
      ANB
      OUT     T96 K10  ; Work    Passage Check OK
6486  LD      T96  ; Work    Passage Check OK
      OUT     T86 D95  ; Rotary  Table ONTime
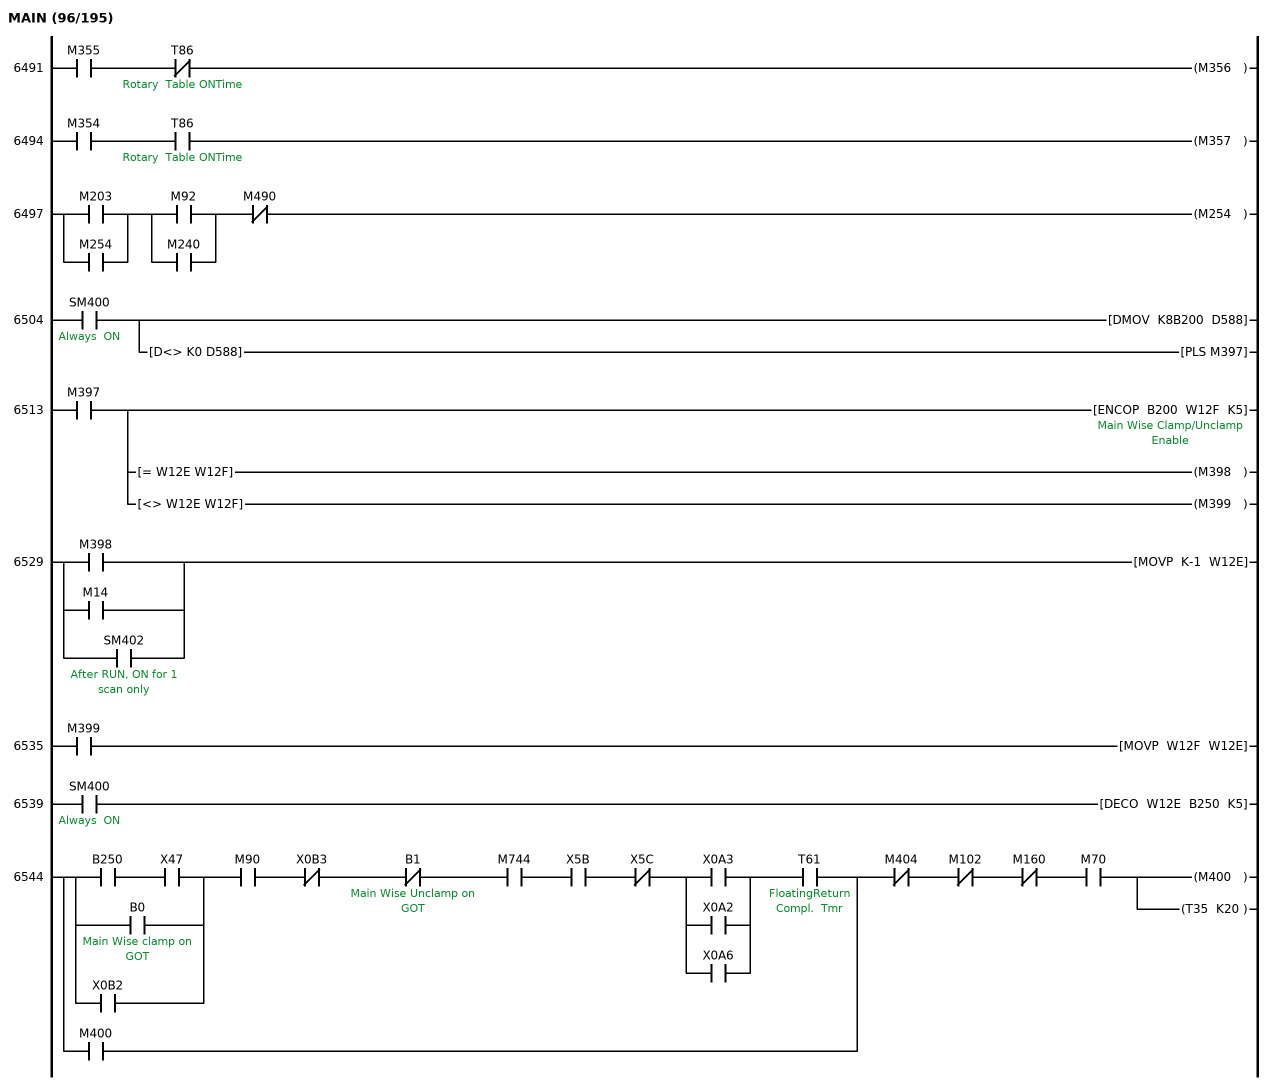
6491  LD      M355
      ANI     T86  ; Rotary  Table ONTime
      OUT     M356
6494  LD      M354
      AND     T86  ; Rotary  Table ONTime
      OUT     M357
6497  LD      M203
      OR      M254
      LD      M92
      OR      M240
      ANB
      ANI     M490
      OUT     M254
6504  LD      SM400  ; Always  ON
      DMOV    K8B200 D588  ; Main Wise Clamp/Unclamp Enable
      ANDD<>  K0 D588
      PLS     M397
6513  LD      M397
      ENCOP   B200 W12F K5
      MPS
      AND=    W12E W12F
      OUT     M398
      MPP
      AND<>   W12E W12F
      OUT     M399
6529  LD      M398
      OR      M14
      OR      SM402  ; After RUN, ON for 1 scan only
      MOVP    K-1 W12E
6535  LD      M399
      MOVP    W12F W12E
6539  LD      SM400  ; Always  ON
      DECO    W12E B250 K5
6544  LD      B250
      AND     X47
      OR      B0  ; Main Wise clamp on GOT
      OR      X0B2
      AND     M90
      ANI     X0B3
      ANI     B1  ; Main Wise Unclamp on GOT
      AND     M744
      AND     X5B
      ANI     X5C
      LD      X0A3
      OR      X0A2
      OR      X0A6
      ANB
      AND     T61  ; FloatingReturn  Compl.  Tmr
      OR      M400
      ANI     M404
      ANI     M102
      ANI     M160
      AND     M70
      OUT     M400
      OUT     T35 K20
